TYPE SensorData :
STRUCT
	force_value_raw AT %I* : REAL;
END_STRUCT
END_TYPE

(* stored: Version 1.1.0.1, ProductVersion 3.1.4024.11
   DUT SensorData: Id {2a92f402-575f-45af-8fd6-9bf206774ea3} *)
